FUNCTION TryConvert_TOD_TO_LINT : BOOL
VAR_INPUT
	in : TOD;
	out : REFERENCE TO LINT;
END_VAR

out := TOD_TO_LINT(in);
TryConvert_TOD_TO_LINT := TRUE;

END_FUNCTION

(* stored: Version 1.1.0.1, ProductVersion 3.1.4024.12
   POU TryConvert_TOD_TO_LINT: Id {f038f0c5-7989-4d89-9a69-d166a9c11496}, SpecialFunc None *)
